// TIA Portal V20 export
DATA_BLOCK "MotorStarterHMI"   // DB212
// stored: MemoryReserve 100
   VAR
      unitMotorstarter : Array[1.."NO_OF_UNITS"] of "typeEmMotorStarterInterface";
   END_VAR
BEGIN
END_DATA_BLOCK
